% RSLogix 500 project DDE MESSANGING_BAK011.RSS, saved by version 8.30.00.16 %
PROJECT "UNTITLED"    % processor: Bul.1763 MicroLogix 1100 Series B %

PROGRAM FILES
  LAD 2   2 rungs
  LAD 3 "CNTR"  10 rungs
  LAD 4 "SYSTEM MOD"  1 rungs

DATA FILES
  O0 OUTPUT  4 elements
  I1 INPUT  6 elements
  S2 STATUS  66 elements
  B3 BINARY  2 elements
  T4 TIMER  1 elements
  C5 COUNTER  1 elements
  R6 CONTROL  1 elements
  N7 INTEGER  6 elements
  F8 FLOAT  10 elements
  ST9 STRING  15 elements

LADDER 2
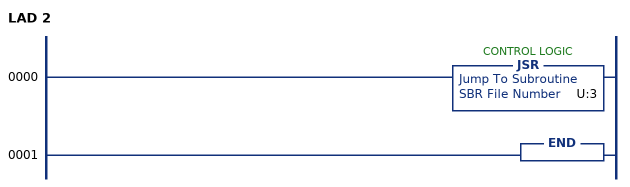
% Rung: 0 %
SOR JSR U:3 EOR
%   U:3  "CONTROL LOGIC" %
% Rung: 1 %
SOR END EOR

LADDER 3 "CNTR"
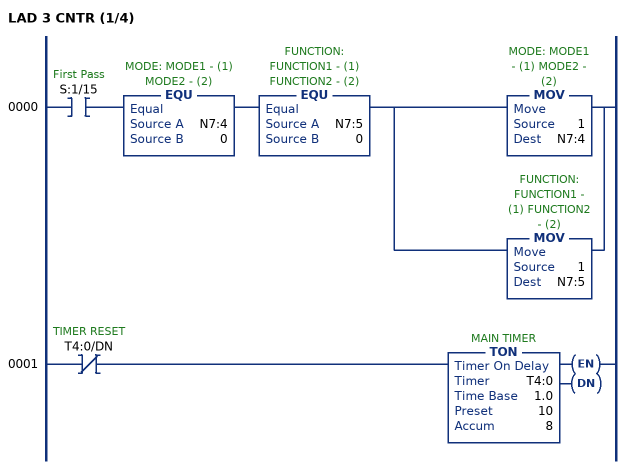
% Rung: 0 %
SOR XIC S:1/15 EQU N7:4 0 EQU N7:5 0 BST MOV 1 N7:4 NXB MOV 1 N7:5 BND EOR
%   S:1/15  "First Pass" %
%   N7:4  "MODE: MODE1 - (1) MODE2 - (2)" %
%   N7:5  "FUNCTION: FUNCTION1 - (1) FUNCTION2 - (2)" %
% Rung: 1 %
SOR XIO T4:0/DN TON T4:0 1.0 10 8 EOR
%   T4:0/DN  "TIMER RESET" %
%   T4:0  "MAIN TIMER" %

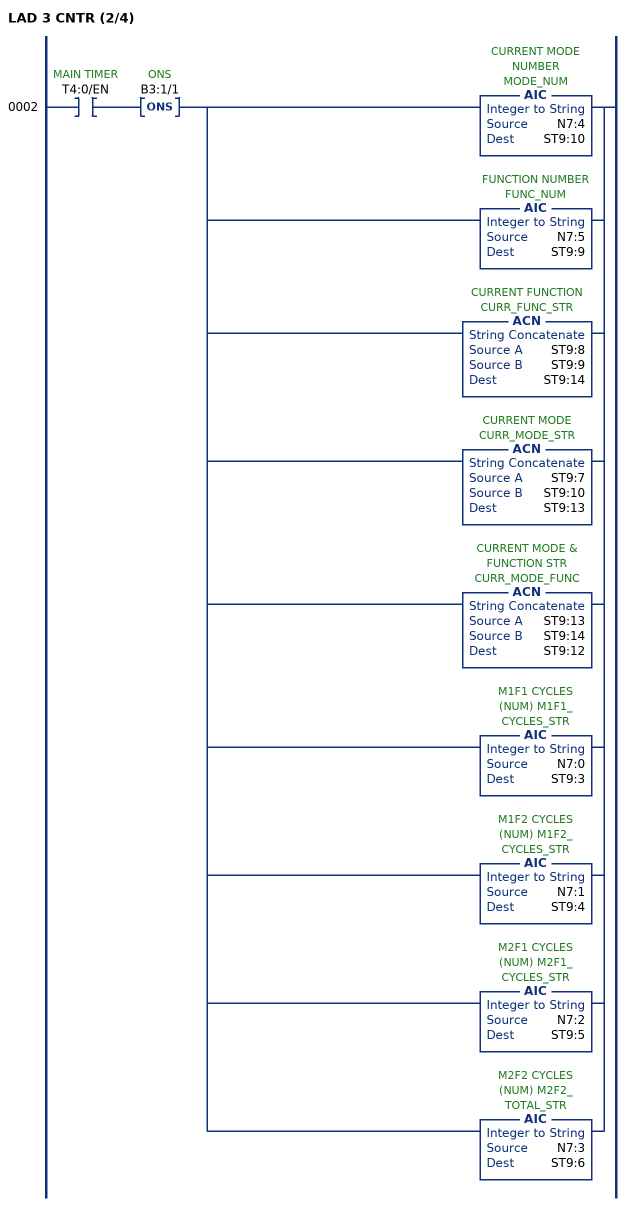
% Rung: 2 %
SOR XIC T4:0/EN ONS B3:1/1 BST AIC N7:4 ST9:10 NXB AIC N7:5 ST9:9 NXB ACN ST9:8 ST9:9 ST9:14 NXB ACN ST9:7 ST9:10 ST9:13 NXB ACN ST9:13 ST9:14 ST9:12 NXB AIC N7:0 ST9:3 NXB AIC N7:1 ST9:4 NXB AIC N7:2 ST9:5 NXB AIC N7:3 ST9:6 BND EOR
%   T4:0  "MAIN TIMER" %
%   B3:1/1  "ONS" %
%   N7:4  "MODE: MODE1 - (1) MODE2 - (2)" %
%   ST9:10  MODE_NUM  "CURRENT MODE NUMBER" %
%   N7:5  "FUNCTION: FUNCTION1 - (1) FUNCTION2 - (2)" %
%   ST9:9  FUNC_NUM  "FUNCTION NUMBER" %
%   ST9:14  CURR_FUNC_STR  "CURRENT FUNCTION" %
%   ST9:13  CURR_MODE_STR  "CURRENT MODE" %
%   ST9:12  CURR_MODE_FUNC  "CURRENT MODE & FUNCTION STR" %
%   N7:0  M1F1_CYCLES  "M1F1 CYCLES COUNTER" %
%   ST9:3  M1F1_CYCLES_STR  "M1F1 CYCLES (NUM)" %
%   N7:1  M1F2_CYCLES  "M1F2 CYCLES COUNTER" %
%   ST9:4  M1F2_CYCLES_STR  "M1F2 CYCLES (NUM)" %
%   N7:2  M2F1_CYCLES  "M2F1 CYCLES COUNTER" %
%   ST9:5  M2F1_CYCLES_STR  "M2F1 CYCLES (NUM)" %
%   N7:3  M2F2_COUNTER  "M2F2 CYCLES COUNTER" %
%   ST9:6  M2F2_TOTAL_STR  "M2F2 CYCLES (NUM)" %

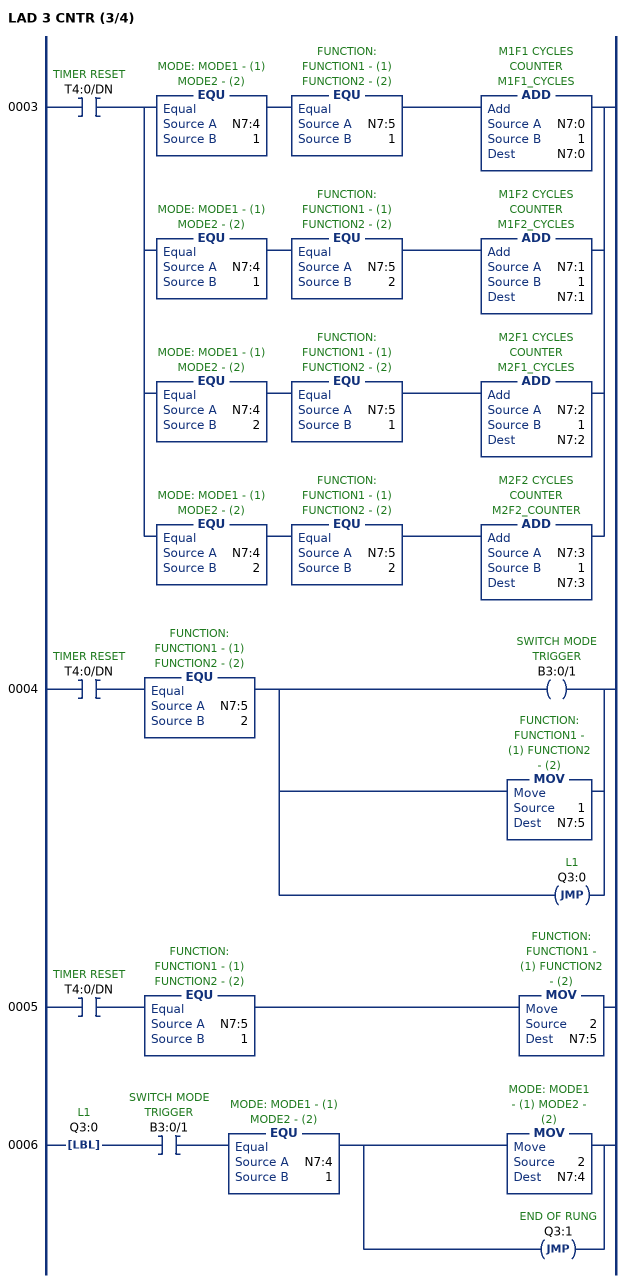
% Rung: 3 %
SOR XIC T4:0/DN BST EQU N7:4 1 EQU N7:5 1 ADD N7:0 1 N7:0 NXB EQU N7:4 1 EQU N7:5 2 ADD N7:1 1 N7:1 NXB EQU N7:4 2 EQU N7:5 1 ADD N7:2 1 N7:2 NXB EQU N7:4 2 EQU N7:5 2 ADD N7:3 1 N7:3 BND EOR
%   T4:0/DN  "TIMER RESET" %
%   N7:4  "MODE: MODE1 - (1) MODE2 - (2)" %
%   N7:5  "FUNCTION: FUNCTION1 - (1) FUNCTION2 - (2)" %
%   N7:0  M1F1_CYCLES  "M1F1 CYCLES COUNTER" %
%   N7:1  M1F2_CYCLES  "M1F2 CYCLES COUNTER" %
%   N7:2  M2F1_CYCLES  "M2F1 CYCLES COUNTER" %
%   N7:3  M2F2_COUNTER  "M2F2 CYCLES COUNTER" %
% Rung: 4 %
SOR XIC T4:0/DN EQU N7:5 2 BST OTE B3:0/1 NXB MOV 1 N7:5 NXB JMP Q3:0 BND EOR
%   T4:0/DN  "TIMER RESET" %
%   N7:5  "FUNCTION: FUNCTION1 - (1) FUNCTION2 - (2)" %
%   B3:0/1  "SWITCH MODE TRIGGER" %
%   Q3:0  "L1" %
% Rung: 5 %
SOR XIC T4:0/DN EQU N7:5 1 MOV 2 N7:5 EOR
%   T4:0/DN  "TIMER RESET" %
%   N7:5  "FUNCTION: FUNCTION1 - (1) FUNCTION2 - (2)" %
% Rung: 6 %
SOR LBL Q3:0 XIC B3:0/1 EQU N7:4 1 BST MOV 2 N7:4 NXB JMP Q3:1 BND EOR
%   Q3:0  "L1" %
%   B3:0/1  "SWITCH MODE TRIGGER" %
%   N7:4  "MODE: MODE1 - (1) MODE2 - (2)" %
%   Q3:1  "END OF RUNG" %

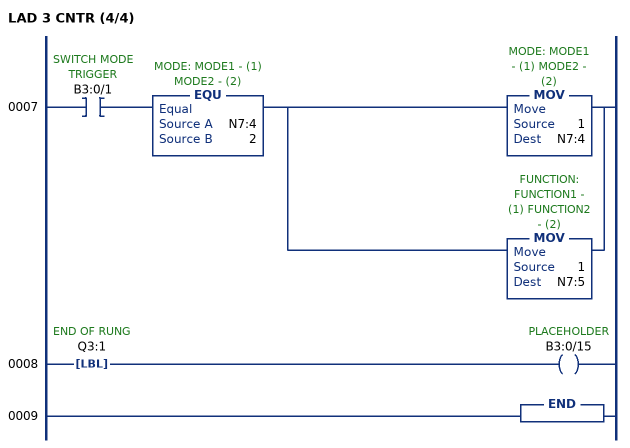
% Rung: 7 %
SOR XIC B3:0/1 EQU N7:4 2 BST MOV 1 N7:4 NXB MOV 1 N7:5 BND EOR
%   B3:0/1  "SWITCH MODE TRIGGER" %
%   N7:4  "MODE: MODE1 - (1) MODE2 - (2)" %
%   N7:5  "FUNCTION: FUNCTION1 - (1) FUNCTION2 - (2)" %
% Rung: 8 %
SOR LBL Q3:1 OTE B3:0/15 EOR
%   Q3:1  "END OF RUNG" %
%   B3:0/15  "PLACEHOLDER" %
% Rung: 9 %
SOR END EOR

OTHER DOCUMENTED ADDRESSES
  ST9:10.0  "MODE NUMBER"
  ST9:11  "CURRENT FUNCTION NUMBER"
  T4:0/1  "MAIN TIMER"

DATA TABLE (non-zero values as saved)
DATA B3
% B3:0 % 0X8000 0X0000
DATA T4
% .PRE .ACC %
% T4:0 % 10 8
DATA N7
% N7:0 % 17 16 16 16 1 2
DATA ST9
% ST9:0 % "CURRENT MODE: "
% ST9:1 % "CURRENT FUNCTION: "
% ST9:2 % "CURRNET MODE + FUNCTION: "
% ST9:3 % "M1F1 TOTAL CYCLES: "
% ST9:4 % "M1F2 TOTAL CYCLES: "
% ST9:5 % "M2F1 TOTAL CYCLES: "
% ST9:6 % "M2F2 TOTAL CYCLES: "
% ST9:7 % "M"
% ST9:8 % "F"
